Yaskawa INFORM job: R1_W63-A1(120,-90)KM-OK_R2.JBI

/JOB
//NAME R1_W63-A1(120,-90)KM-OK_R2
///FOLDERNAME KRIS-SCIANA
//POS
///NPOS 37,37,0,3,0,0
///TOOL 0
///POSTYPE PULSE
///PULSE
C00000=-15507,74076,-2347,-18134,100161,88161
C00001=-20171,3250,-42059,-16045,87905,88501
C00002=-44846,-16350,-36708,26928,67857,83216
C00003=-29722,-6489,-18602,20815,57983,87106
C00004=-29722,-6380,-17141,21001,57194,86947
C00005=-29722,-6393,-17284,20983,57270,86963
C00006=-29722,-6393,-17284,20983,57270,86963
C00007=-28274,-7679,-18312,20209,56882,87496
C00008=-28905,-7260,-19785,20308,58092,87470
C00009=-28905,-7239,-26034,19567,61726,88152
C00010=-64788,-94726,-75227,38489,61488,72518
C00011=112115,62983,54736,-4036,72204,-8101
C00012=-65809,-96957,-70344,40235,58702,70845
C00013=-65809,-96262,-68916,40437,58299,70667
C00014=-65809,-96346,-69089,40411,58347,70688
C00015=-62987,-100350,-70529,40163,56144,71145
C00016=-65227,-97943,-70899,40148,58306,70966
C00017=-35648,-33433,-51629,581,106969,87586
C00018=-36431,-36585,-53684,531,106624,87314
C00019=-35362,-32257,-50845,597,107094,87687
C00020=-42999,-25077,-43525,9882,111826,86220
C00021=-52034,-15572,-30579,21796,117162,85059
C00022=158501,49549,56228,-16946,45407,14810
C00023=158535,50209,58031,-17189,44676,14967
C00024=-75499,-44012,-36379,52113,95484,71575
C00025=-63711,-26814,-25221,52577,89998,74800
C00026=-51755,270,-4453,52122,83926,77656
C00027=-45821,31942,27037,51972,78603,77811
C00028=-42474,24679,26787,59593,60621,74916
C00029=-41984,26974,29022,59607,60212,74927
C00030=-43138,19505,16213,57996,63097,76469
C00031=-26305,1577,-38700,13145,85063,89178
C00032=2719,6086,-32804,8720,83267,77624
C00033=11495,132223,115006,11835,51584,66229
C00034=11117,131903,115148,12421,51473,61966
C00035=30495,213544,175638,12421,51473,61966
C00036=29280,212341,155928,12421,51473,61966
BC00000=114698,5829,1017531
BC00001=114698,5829,1017531
BC00002=114698,5829,882926
BC00003=114698,5829,882926
BC00004=114698,5829,882926
BC00005=114698,5829,882926
BC00006=114698,5829,882926
BC00007=114698,5829,882926
BC00008=114698,5829,882926
BC00009=114698,5829,882926
BC00010=114698,5829,882926
BC00011=322254,371612,1073831
BC00012=114698,5829,882926
BC00013=114698,5829,882926
BC00014=114698,5829,882926
BC00015=114698,5829,882926
BC00016=114698,5829,882926
BC00017=114698,5829,882926
BC00018=114698,5829,882926
BC00019=114698,5829,882926
BC00020=114780,5930,882979
BC00021=114698,5829,882926
BC00022=398174,356867,1075175
BC00023=398174,356867,1075175
BC00024=114698,5829,882926
BC00025=114698,5829,882926
BC00026=114908,6089,883061
BC00027=101107,64,898017
BC00028=101107,64,898017
BC00029=101107,64,898017
BC00030=101107,64,898017
BC00031=101107,64,898017
BC00032=154974,2765,927803
BC00033=77675,67272,944379
BC00034=77600,26253,951400
BC00035=77600,26253,1018775
BC00036=77600,552091,1026125
///POSTYPE BASE
///RECTAN
///RCONF 0,0,0,0,1,0,0,0,0,0,0,0,0,0,0,0,0,0,0,0,0,0,0,0
P00006=2.006,1.622,-0.565,0.0000,0.0000,0.0000
P00021=0.073,2.058,-0.109,0.0000,0.0000,0.0000
P00022=2.006,1.622,-0.565,0.0000,0.0000,0.0000
//INST
///DATE 2025/04/14 11:19
///ATTR SC,RW
///GROUP1 RB1,BS1
NOP
'Path S1152
SFTOF
MOVJ C00000 BC00000 VJ=20.00
MOVJ C00001 BC00001 VJ=20.00
MOVL C00002 BC00002 V=100.0
MOVL C00003 BC00003 V=60.0
REFP 3 C00004 BC00004
CALL JOB:SEARCH-R1
SET P021 P006
SFTON P021
MOVL C00005 BC00005 V=60.0
MOVL C00006 BC00006 V=60.0
REFP 3 C00007 BC00007
CALL JOB:SEARCH-R1
SET P021 P006
SFTON P021
MOVL C00008 BC00008 V=60.0
SFTOF
MOVL C00009 BC00009 V=100.0
MOVL C00010 BC00010 V=100.0
'Path S1153
SFTOF
COMM MOVJ C00011 BC00011 VJ=20.00
MOVL C00012 BC00012 V=100.0
REFP 3 C00013 BC00013
CALL JOB:SEARCH-R1
SET P022 P006
SFTON P022
MOVL C00014 BC00014 V=60.0
REFP 3 C00015 BC00015
CALL JOB:SEARCH-R1
SET P022 P006
SFTON P022
MOVL C00016 BC00016 V=60.0
MOVL C00017 BC00017 V=100.0
REFP 3 C00018 BC00018
CALL JOB:SEARCH-R1
SET P022 P006
SFTON P022
MOVL C00019 BC00019 V=60.0
'Path W1154
SFTOF
SFTON P022
CALL JOB:COFNIJ_DRUT
MOVL C00020 BC00020 V=100.0
MOVL C00021 BC00021 V=100.0 PL=0
REFP 1 C00022 BC00022
REFP 2 C00023 BC00023
MACRO1 MJ#(0) ARGF9
ARCON
MOVL C00024 BC00024 V=11.7
MOVL C00025 BC00025 V=11.7
SFTON P021
MOVL C00026 BC00026 V=11.7
MOVL C00027 BC00027 V=11.7
MOVL C00028 BC00028 V=11.7
MOVL C00029 BC00029 V=11.7
ARCOF
MOVL C00030 BC00030 V=100.0
MOVL C00031 BC00031 V=200.0
SFTOF
MOVJ C00032 BC00032 VJ=20.00
MOVJ C00033 BC00033 VJ=20.00
MOVJ C00034 BC00034 VJ=100.00
MOVJ C00035 BC00035 VJ=100.00
MOVJ C00036 BC00036 VJ=100.00
SFTOF
END
